// TIA Portal V21 export
FUNCTION "FC_Conveyor_sides" : Void   // FC4, LAD
TITLE = Control de Cintas Laterales
{ S7_Optimized_Access := 'TRUE' }
// stored: SetENOAutomatically false
   VAR_INPUT
      Emergencia : Bool;
      "Sistema en marcha" : Bool;
   END_VAR
   VAR_OUTPUT
      "Conveyor left" : Bool;
      "Conveyor right" : Bool;
   END_VAR
BEGIN

REGION Network 1: Activacion/Desactivacion de cintas laterales
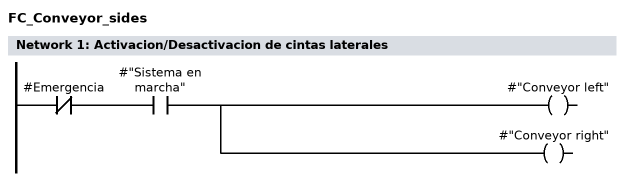
   RUNG wire#powerrail
      I_Contact( #Emergencia )
      Contact( #"Sistema en marcha" )
      wire#w1
      Coil( #"Conveyor left" )
   END_RUNG
   RUNG wire#w1
      Coil( #"Conveyor right" )
   END_RUNG
   // the same network as SCL:
   #"Conveyor left" := NOT #Emergencia AND #"Sistema en marcha";
   #"Conveyor right" := #"Conveyor left";
END_REGION
END_FUNCTION
